(* IEC 61131-3 sources: POMIRTS_lab3/AS/Library/AsNetX, 2 files *)

(* ---- AsNetX.fun ---- *)
(********************************************************************
 * COPYRIGHT -- Bernecker + Rainer
 ********************************************************************
 * Library: AsNetX
 * File: AsNetX.fun
 * Author: B+R
 ********************************************************************
 * Functions and function blocks of library AsNetX
 ********************************************************************)

FUNCTION_BLOCK netxConfig				(*download configuration*)
	VAR_INPUT
		enable			: BOOL;			(*enables execution*)
		pDevice			: UDINT;		(*pointer to the device name*)
		pConfig			: UDINT;		(*pointer to the configuration name*)
	END_VAR

	VAR_OUTPUT
		status			: UINT;			(*execution status: ERR_OK, ERR_FUB_ENABLE_FALSE, ERR_FUB_BUSY, 0xXXXX = see help*)
		ident			: UDINT;		(*handle for further use*)
	END_VAR

	VAR
        i_state			: UINT;			(*internal variable*)
		i_result		: UINT;			(*internal variable*)
        i_tmp			: UDINT;		(*internal variable*)
	END_VAR
END_FUNCTION_BLOCK

FUNCTION_BLOCK netxXConfig				(*download configuration*)
	VAR_INPUT
		enable			: BOOL;			(*enables execution*)
		pDevice			: UDINT;		(*pointer to the device name*)
		pConfig			: UDINT;		(*pointer to the configuration name*)
		flags			: UDINT;		(*flags*)
	END_VAR

	VAR_OUTPUT
		status			: UINT;			(*execution status: ERR_OK, ERR_FUB_ENABLE_FALSE, ERR_FUB_BUSY, 0xXXXX = see help*)
		ident			: UDINT;		(*handle for further use*)
	END_VAR

	VAR
        i_state			: UINT;			(*internal variable*)
		i_result		: UINT;			(*internal variable*)
        i_tmp			: UDINT;		(*internal variable*)
	END_VAR
END_FUNCTION_BLOCK

FUNCTION_BLOCK netxStart				(*start communication*)
	VAR_INPUT
		enable			: BOOL;			(*enables execution*)
		ident			: UDINT;		(*handle*)
	END_VAR

	VAR_OUTPUT
		status			: UINT;			(*execution status: ERR_OK, ERR_FUB_ENABLE_FALSE, ERR_FUB_BUSY, 0xXXXX = see help*)
	END_VAR

	VAR
        i_state			: UINT;			(*internal variable*)
		i_result		: UINT;			(*internal variable*)
        i_tmp			: UDINT;		(*internal variable*)
	END_VAR
END_FUNCTION_BLOCK

FUNCTION_BLOCK netxStop				(*stop communication*)
	VAR_INPUT
		enable			: BOOL;			(*enables execution*)
		ident			: UDINT;		(*handle*)
	END_VAR

	VAR_OUTPUT
		status			: UINT;			(*execution status: ERR_OK, ERR_FUB_ENABLE_FALSE, ERR_FUB_BUSY, 0xXXXX = see help*)
	END_VAR

	VAR
        i_state			: UINT;			(*internal variable*)
		i_result		: UINT;			(*internal variable*)
        i_tmp			: UDINT;		(*internal variable*)
	END_VAR
END_FUNCTION_BLOCK

FUNCTION_BLOCK netxIORdWr				(*exchange IO data*)
	VAR_INPUT
		enable			: BOOL;			(*enables execution*)
		ident			: UDINT;		(*handle*)
		pIn				: UDINT;		(*pointer to the input data*)
		inArea			: UDINT;		(*area of input  data*)
		inOffset		: UDINT;		(*offset of input  data*)
		inSize			: UDINT;		(*size of input  data*)
		pOut			: UDINT;		(*pointer to the output data*)
		outArea			: UDINT;		(*area of output  data*)
		outOffset		: UDINT;		(*offset of output  data*)
		outSize			: UDINT;		(*size of output datd*)
	END_VAR

	VAR_OUTPUT
		status			: UINT;			(*execution status: ERR_OK, 0xXXXX = see help*)
	END_VAR
END_FUNCTION_BLOCK

FUNCTION_BLOCK netxDpSAdrSet			(*set profibus slave address*)
	VAR_INPUT
		enable			: BOOL;			(*enables execution*)
		ident			: UDINT;		(*handle*)
		address			: UDINT;		(*address*)
	END_VAR

	VAR_OUTPUT
		status			: UINT;			(*execution status: ERR_OK, ERR_FUB_ENABLE_FALSE, ERR_FUB_BUSY, 0xXXXX = see help*)
		dpStatus		: UDINT;		(*profibus DP stack status*)
	END_VAR

	VAR
        i_state			: UINT;			(*internal variable*)
		i_result		: UINT;			(*internal variable*)
        i_tmp			: UDINT;		(*internal variable*)
	END_VAR
END_FUNCTION_BLOCK

(* ---- AsNetX.var ---- *)
(********************************************************************
 * COPYRIGHT -- Bernecker + Rainer
 ********************************************************************
 * Library: AsNetX
 * File: AsNetX.var
 * Author: B+R
 ********************************************************************
 * Local variables of library AsNetX
 ********************************************************************)

VAR CONSTANT
	netxERR_DEVICE				: UINT := 35001;	(*device error*)
	netxERR_IDENT				: UINT := 35002;	(*ident error*)
	netxERR_DRV_OPEN			: UINT := 35003;	(*open driver error*)
	netxERR_SYSDEV_OPEN			: UINT := 35004;	(*open sysdevice error*)
	netxERR_CFG_MODULE			: UINT := 35005;	(*configuration module error*)
	netxERR_CFG_DOWNLOAD		: UINT := 35006;	(*configuration download error*)
	netxERR_CHANNEL_OPEN		: UINT := 35007;	(*open channel error*)
	netxERR_RESET				: UINT := 35008;	(*reset error*)
	netxERR_SET_STATE			: UINT := 35009;	(*communication start/stop error*)
	netxERR_BUS_STATE			: UINT := 35010;	(*communication bus state error*)
	netxERR_IO_READ				: UINT := 35011;	(*read io error*)
	netxERR_IO_WRITE			: UINT := 35012;	(*write io error*)
	netxERR_PACKET				: UINT := 35013;	(*put/get packet error*)
	netxERR_STACK				: UINT := 35014;	(*stack error*)

	netxSTART_BY_USER			: UDINT	:= 16#00000001;	(*bus communication started by user*)
END_VAR
